(* PLC project  *)

CONFIGURATION MR_J5_G_RJN1
END_CONFIGURATION
